SUBAPPLICATION Uebung_004b (* Toggle Flip-Flop mit IE / E_SWITCH + E_SR *)
  (* Standard: 61499-2; Description: Copyright (c) 2023 Meisterschulen am Ostbahnhof This program and the accompanying materials are made available under the terms of the Eclipse Public License 2.0 which is available at https://www.eclipse.org/legal/epl-2.0/ SPDX-License-Identifier: EPL-2.0 *)
  (* Version 1.0, 2023-10-23, Franz Höpfinger, Meisterschulen am Ostbahnhof *)
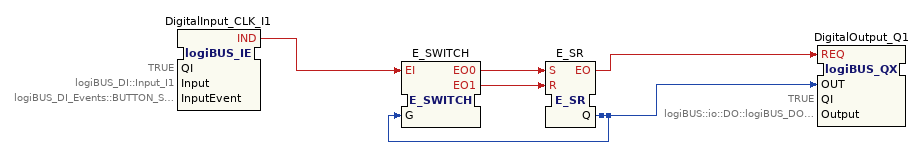
  FBS
    DigitalOutput_Q1 : logiBUS_QX(QI := TRUE, Output := logiBUS::io::DO::logiBUS_DO::Output_Q1);
    DigitalInput_CLK_I1 : logiBUS_IE(QI := TRUE, Input := logiBUS_DI::Input_I1, InputEvent := logiBUS_DI_Events::BUTTON_SINGLE_CLICK);
    E_SR : E_SR;
    E_SWITCH : E_SWITCH;
  END_FBS
  EVENT_CONNECTIONS
    E_SR.EO TO DigitalOutput_Q1.REQ;
    E_SWITCH.EO0 TO E_SR.S;
    E_SWITCH.EO1 TO E_SR.R;
    DigitalInput_CLK_I1.IND TO E_SWITCH.EI;
  END_CONNECTIONS
  DATA_CONNECTIONS
    E_SR.Q TO DigitalOutput_Q1.OUT;
    E_SR.Q TO E_SWITCH.G;
  END_CONNECTIONS
END_SUBAPPLICATION
